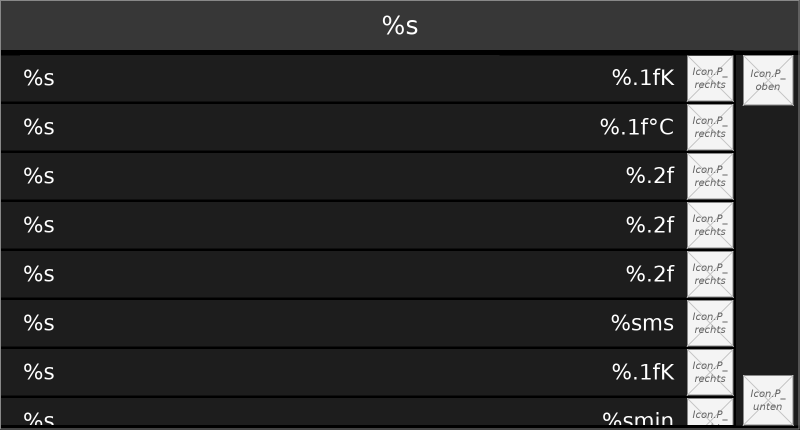
VISUALIZATION SW_WP_EEV_Liste  // 800x430
VAR_IN_OUT
	FB_EEV:EEV;	
	
END_VAR
	
VAR_INPUT
	i_Titel:INT;

END_VAR

VAR
	i_ref_versch:INT;
END_VAR
    Rectangle (0,0 800x50), "%s", text list: 'Sprachen', text index: i_Titel
    Rectangle (736,55 64x370)
    Image (743,375 50x50), image: Icon.P_unten
        OnMouseClick: execute { i_ref_versch:=i_ref_versch + 53; }
    Image (743,55 50x50), image: Icon.P_oben
        OnMouseClick: execute { i_ref_versch:=i_ref_versch - 53; }
    Group (0,50 733x590)
        p2738717112: i_ref_versch
        Rectangle (0,5 733x46)
        Rectangle (0,54 733x46)
        Rectangle (547,5 130x45), "%.1fK", text variable: FB_EEV.f_SollwertUBH
        Rectangle (547,54 130x46), "%.1f°C", text variable: FB_EEV.f_MOP
        Image (687,5 46x46), image: Icon.P_rechts
            OnMouseClick: execute { GWP_Library.Visu.i_Frame_Index:=1; }
        Image (687,54 46x46), image: Icon.P_rechts
            OnMouseClick: execute { GWP_Library.Visu.i_Frame_Index:=2; }
        Rectangle (0,103 733x46)
        Rectangle (0,152 733x46)
        Rectangle (0,201 733x46)
        Rectangle (0,250 733x46)
        Rectangle (0,299 733x46)
        Rectangle (0,348 733x46)
        Rectangle (0,397 733x46)
        Rectangle (0,446 733x46)
        Rectangle (0,495 733x46)
        Rectangle (547,103 130x45), "%.2f", text variable: FB_EEV.f_PFaktor
            OnMouseClick: execute { GWP_Library.Visu.i_Frame_Index:=2; }
        Rectangle (547,152 130x46), "%.2f", text variable: FB_EEV.f_IFaktor
        Rectangle (547,201 130x46), "%.2f", text variable: FB_EEV.f_DFaktor
        Rectangle (547,250 130x46), "%sms", text variable: FB_EEV.t_Takt.wMilliseconds
        Rectangle (547,299 130x46), "%.1fK", text variable: FB_EEV.f_MinUBH
        Rectangle (547,348 130x46), "%smin", text variable: FB_EEV.t_AL_EEV.wMinute
        Rectangle (547,446 130x46), "Ein"
        Rectangle (547,495 130x46), "Ein"
        Image (687,103 46x46), image: Icon.P_rechts
            OnMouseClick: execute { GWP_Library.Visu.i_Frame_Index:=3; }
        Image (687,495 46x46), image: Icon.P_rechts
        Image (687,446 46x46), image: Icon.P_rechts
        Image (687,397 46x46), image: Icon.P_rechts
            OnMouseClick: execute { GWP_Library.Visu.i_Frame_Index:=9; }
        Image (687,348 46x46), image: Icon.P_rechts
            OnMouseClick: execute { GWP_Library.Visu.i_Frame_Index:=8; }
        Image (687,299 46x46), image: Icon.P_rechts
            OnMouseClick: execute { GWP_Library.Visu.i_Frame_Index:=7; }
        Image (687,250 46x46), image: Icon.P_rechts
            OnMouseClick: execute { GWP_Library.Visu.i_Frame_Index:=6; }
        Image (687,201 46x46), image: Icon.P_rechts
            OnMouseClick: execute { GWP_Library.Visu.i_Frame_Index:=5; }
        Image (687,152 46x46), image: Icon.P_rechts
            OnMouseClick: execute { GWP_Library.Visu.i_Frame_Index:=4; }
        Rectangle (0,544 733x46)
        Rectangle (547,544 130x45), "Ein"
        Image (687,544 46x46), image: Icon.P_rechts
        Image (79,380 50x50), image: Icon.zurueck
            OnMouseClick:  Assign=Sollwertmenu_Waermegewinnung, Type=Assignment
            OnMouseClick: execute { i_verschieben:=0; }
        Rectangle (0,0 733x5)
        Rectangle (20,5 479x46), "%s", text list: 'Sprachen', text index: 85
        Rectangle (20,54 479x46), "%s", text list: 'Sprachen', text index: 86
        Rectangle (20,152 479x46), "%s", text list: 'Sprachen', text index: 88
        Rectangle (20,103 479x46), "%s", text list: 'Sprachen', text index: 87
        Rectangle (20,201 479x46), "%s", text list: 'Sprachen', text index: 89
        Rectangle (20,250 479x46), "%s", text list: 'Sprachen', text index: 90
        Rectangle (20,299 479x46), "%s", text list: 'Sprachen', text index: 91
        Rectangle (20,348 479x46), "%s", text list: 'Sprachen', text index: 92
        Rectangle (20,397 479x46), "%s", text list: 'Sprachen', text index: 72
        Rectangle (20,446 479x46), "%s", text list: 'Sprachen'
        Rectangle (20,495 479x46), "%s", text list: 'Sprachen'
        Rectangle (20,544 479x46), "%s", text list: 'Sprachen'
        Rectangle (0,375 733x5)
END_VISUALIZATION

// VISUs/Sollwertmenu_9/Wärmepumpe/Einsatzgrenzen/SW_WP_Einsatzgrenzen
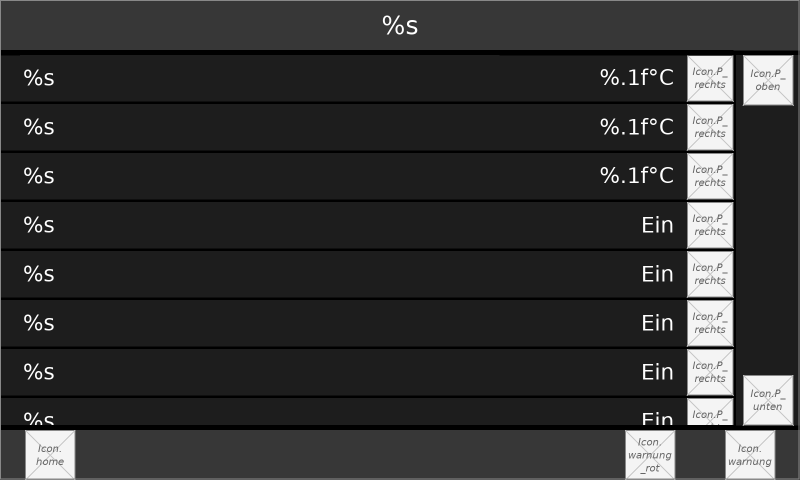
VISUALIZATION SW_WP_Einsatzgrenzen  // 800x480
VAR_IN_OUT
	FB_Einsatzgrenzen:Einsatzgrenzen;
END_VAR
    Frame (0,0 800x430)
        shows SW_WP_Einsatzgrenzen_Liste()
    Frame (0,430 800x50)
        shows Fusszeile_50()
END_VISUALIZATION

// VISUs/Sollwertmenu_9/Wärmepumpe/Einsatzgrenzen/SW_WP_Einsatzgrenzen_Liste
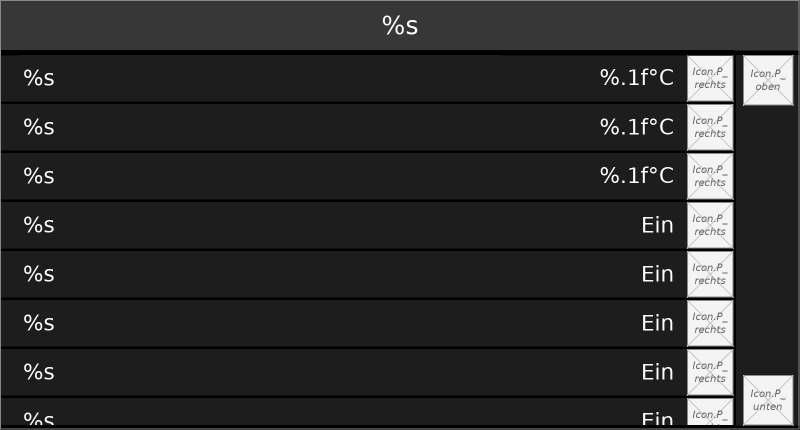
VISUALIZATION SW_WP_Einsatzgrenzen_Liste  // 800x430
VAR_IN_OUT
	FB_Einsatzgrenzen:Einsatzgrenzen;
END_VAR

VAR_INPUT
	i_Titel:INT;
END_VAR

VAR
	i_verschieben:INT;
 END_VAR
    Rectangle (0,55 733x46)
    Rectangle (0,104 733x46)
    Rectangle (547,55 130x45), "%.1f°C", text variable: FB_EEV.f_Regelsignal
    Rectangle (547,104 130x46), "%.1f°C"
    Image (687,55 46x46), image: Icon.P_rechts
        OnMouseClick: execute { GWP_Library.Visu.i_Frame_Index:=1; }
    Image (687,104 46x46), image: Icon.P_rechts
        OnMouseClick: execute { GWP_Library.Visu.i_Frame_Index:=2; }
    Rectangle (0,153 733x46)
    Rectangle (0,202 733x46)
    Rectangle (0,251 733x46)
    Rectangle (0,300 733x46)
    Rectangle (0,349 733x46)
    Rectangle (0,398 733x46)
    Rectangle (0,447 733x46)
    Rectangle (0,496 733x46)
    Rectangle (0,545 733x46)
    Rectangle (547,153 130x45), "%.1f°C"
        OnMouseClick: execute { GWP_Library.Visu.i_Frame_Index:=2; }
    Rectangle (547,202 130x46), "Ein"
    Rectangle (547,251 130x46), "Ein"
    Rectangle (547,300 130x46), "Ein"
    Rectangle (547,349 130x46), "Ein"
    Rectangle (547,447 130x46), "Ein"
    Rectangle (547,398 130x46), "Ein"
    Rectangle (547,496 130x46), "Ein"
    Rectangle (547,545 130x46), "Ein"
    Image (687,153 46x46), image: Icon.P_rechts
        OnMouseClick: execute { GWP_Library.Visu.i_Frame_Index:=3; }
    Image (687,545 46x46), image: Icon.P_rechts
    Image (687,496 46x46), image: Icon.P_rechts
    Image (687,447 46x46), image: Icon.P_rechts
    Image (687,398 46x46), image: Icon.P_rechts
    Image (687,349 46x46), image: Icon.P_rechts
    Image (687,300 46x46), image: Icon.P_rechts
    Image (687,251 46x46), image: Icon.P_rechts
    Image (687,202 46x46), image: Icon.P_rechts
    Rectangle (0,594 733x46)
    Rectangle (547,594 130x45), "Ein"
    Image (687,594 46x46), image: Icon.P_rechts
    Image (79,430 50x50), image: Icon.zurueck
        OnMouseClick:  Assign=Sollwertmenu_Waermegewinnung, Type=Assignment
        OnMouseClick: execute { i_verschieben:=0; }
    Rectangle (0,0 800x50), "%s", text list: 'Sprachen', text index: i_Titel
    Rectangle (736,55 64x370)
    Image (743,375 50x50), image: Icon.P_unten
        OnMouseClick: execute {
            IF i_verschieben<0 THEN
            	i_verschieben:=i_verschieben+53;
            End_if
        }
    Image (743,55 50x50), image: Icon.P_oben
        OnMouseClick: execute {
            IF  i_verschieben>-200 THEN
            	i_verschieben:=i_verschieben-53;
            End_if
        }
    Rectangle (0,50 733x5)
    Rectangle (20,55 479x46), "%s", text list: 'Sprachen'
    Rectangle (20,104 479x46), "%s", text list: 'Sprachen'
    Rectangle (20,202 479x46), "%s", text list: 'Sprachen'
    Rectangle (20,153 479x46), "%s", text list: 'Sprachen'
    Rectangle (20,251 479x46), "%s", text list: 'Sprachen'
    Rectangle (20,300 479x46), "%s", text list: 'Sprachen'
    Rectangle (20,349 479x46), "%s", text list: 'Sprachen'
    Rectangle (20,398 479x46), "%s", text list: 'Sprachen'
    Rectangle (20,447 479x46), "%s", text list: 'Sprachen'
    Rectangle (20,496 479x46), "%s", text list: 'Sprachen'
    Rectangle (20,545 479x46), "%s", text list: 'Sprachen'
    Rectangle (20,594 479x46), "%s", text list: 'Sprachen'
    Rectangle (0,425 733x5)
END_VISUALIZATION

// VISUs/Sollwertmenu_9/Wärmepumpe/Kachel_Allgemein
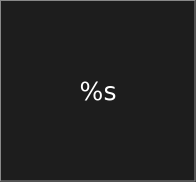
VISUALIZATION Kachel_Allgemein  // 196x182
    Rectangle (0,0 196x182), "%s", text list: 'Sprachen', text index: 18
END_VISUALIZATION

// VISUs/Sollwertmenu_9/Wärmepumpe/Kachel_EEV
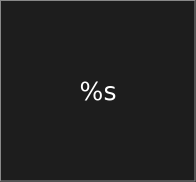
VISUALIZATION Kachel_EEV  // 196x182
    Rectangle (0,0 196x182), "%s", text list: 'Sprachen', text index: 15
END_VISUALIZATION

// VISUs/Sollwertmenu_9/Wärmepumpe/Kachel_Einsatzgrenzen
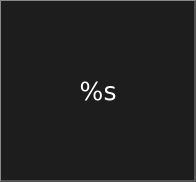
VISUALIZATION Kachel_Einsatzgrenzen  // 196x182
    Rectangle (0,0 196x182), "%s", text list: 'Sprachen', text index: 16
END_VISUALIZATION

// VISUs/Sollwertmenu_9/Wärmepumpe/Kachel_Verdichter
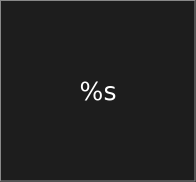
VISUALIZATION Kachel_Verdichter  // 196x182
    Rectangle (0,0 196x182), "%s", text list: 'Sprachen', text index: 17
END_VISUALIZATION

// VISUs/Sollwertmenu_9/Wärmepumpe/Sollwertmenu_Waermepumpe
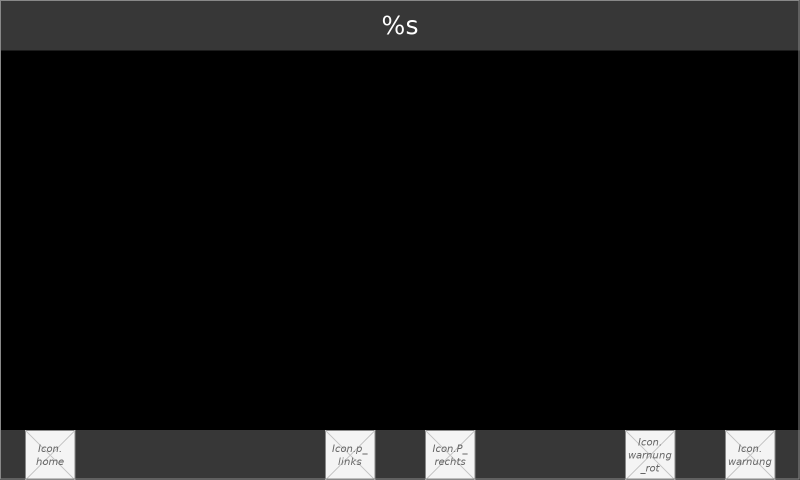
VISUALIZATION Sollwertmenu_Waermepumpe  // 800x480
VAR_IN_OUT
		
END_VAR

VAR
	i_verschieben:INT;

END_VAR
    Image (425,430 50x50), image: Icon.reinnavigieren
    Image (325,430 50x50), image: Icon.reinnavigieren
    Rectangle (0,0 800x50), "%s", text list: 'Sprachen', text index: 14
    Frame (0,430 800x50)
        shows Fusszeile_50()
    Image (425,430 50x50), image: Icon.P_rechts
        OnMouseClick: execute {
            IF i_verschieben>-800 THEN
            	i_verschieben:=i_verschieben-800;
            END_IF
        }
    Image (325,430 50x50), image: Icon.p_links
        OnMouseClick: execute {
            IF i_verschieben<0 THEN
            	i_verschieben:=i_verschieben+800;
            END_IF
        }
    Rectangle (88,515 454x57), "Kachel 1: 0;55 *** Kachel 2: 201;55 *** Kachel 3: 402;55 *** Kachel 4: 604;55 Kachel 5: 0;242 *** Kachel 6: 201;242 *** Kachel 7: 402;242 *** Kachel 8: 604;242"
END_VISUALIZATION

// VISUs/Sollwertmenu_9/Wärmesenke/Kachel_Heizgruppen
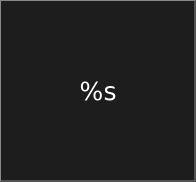
VISUALIZATION Kachel_Heizgruppen  // 196x182
    Rectangle (0,0 196x182), "%s", text list: 'Sprachen', text index: 23
END_VISUALIZATION

// VISUs/Sollwertmenu_9/Wärmesenke/Kachel_Hochhaltung
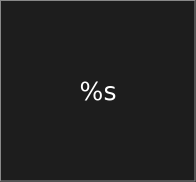
VISUALIZATION Kachel_Hochhaltung  // 196x182
    Rectangle (0,0 196x182), "%s", text list: 'Sprachen', text index: 24
END_VISUALIZATION

// VISUs/Sollwertmenu_9/Wärmesenke/Kachel_HWP
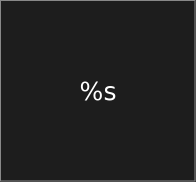
VISUALIZATION Kachel_HWP  // 196x182
    Rectangle (0,0 196x182), "%s", text list: 'Sprachen', text index: 21
END_VISUALIZATION

// VISUs/Sollwertmenu_9/Wärmesenke/Kachel_TWW
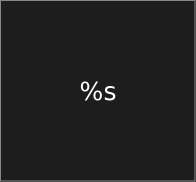
VISUALIZATION Kachel_TWW  // 196x182
    Rectangle (0,0 196x182), "%s", text list: 'Sprachen', text index: 22
END_VISUALIZATION

// VISUs/Sollwertmenu_9/Wärmesenke/Kachel_UWP_Verfl
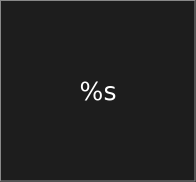
VISUALIZATION Kachel_UWP_Verfl  // 196x182
    Rectangle (0,0 196x182), "%s", text list: 'Sprachen', text index: 20
END_VISUALIZATION

// VISUs/Sollwertmenu_9/Wärmesenke/Sollwertmenu_Waermesenke
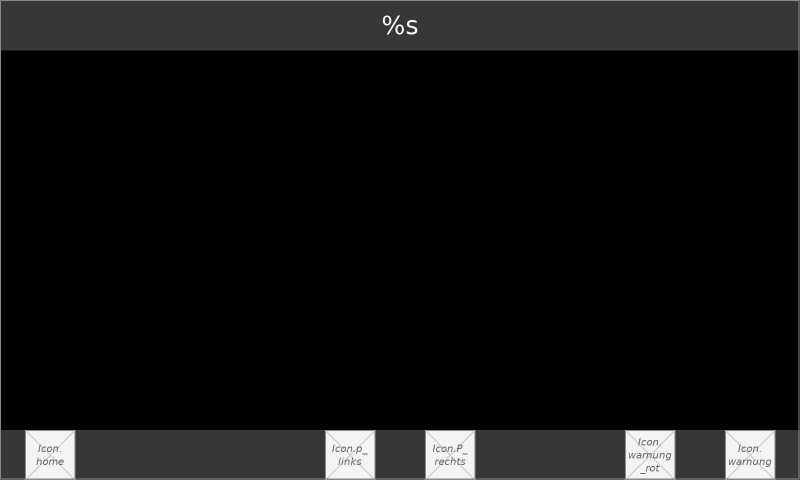
VISUALIZATION Sollwertmenu_Waermesenke  // 800x480
VAR_IN_OUT
		
END_VAR

VAR
	i_verschieben:INT;

END_VAR
    Image (425,430 50x50), image: Icon.reinnavigieren
    Image (325,430 50x50), image: Icon.reinnavigieren
    Rectangle (0,0 800x50), "%s", text list: 'Sprachen', text index: 19
    Frame (0,430 800x50)
        shows Fusszeile_50()
    Image (425,430 50x50), image: Icon.P_rechts
        OnMouseClick: execute {
            IF i_verschieben>-800 THEN
            	i_verschieben:=i_verschieben-800;
            END_IF
        }
    Image (325,430 50x50), image: Icon.p_links
        OnMouseClick: execute {
            IF i_verschieben<0 THEN
            	i_verschieben:=i_verschieben+800;
            END_IF
        }
    Rectangle (88,515 483x57), "Kachel 1: 0;55 *** Kachel 2: 201;55 *** Kachel 3: 402;55 *** Kachel 4: 604;55 Kachel 5: 0;242 *** Kachel 6: 201;242 *** Kachel 7: 402;242 *** Kachel 8: 604;242"
END_VISUALIZATION

// VISUs/Sprache/Spracheistellungen
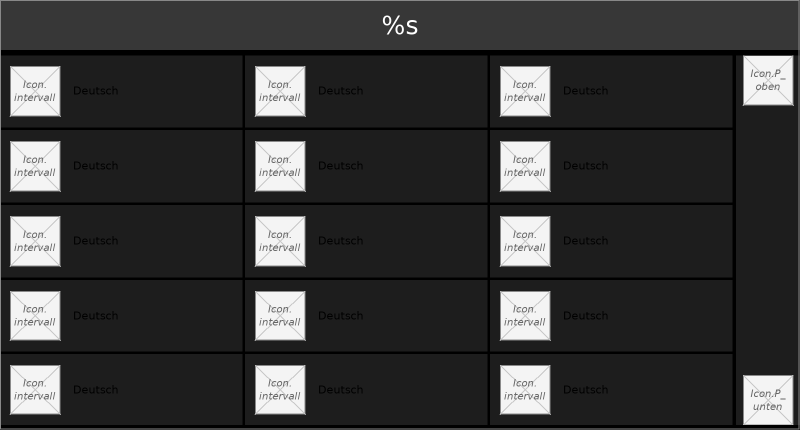
VISUALIZATION Spracheistellungen  // 800x430
VAR_IN_OUT

END_VAR

VAR_INPUT
	
END_VAR

VAR
	i_verschieben:INT;
 END_VAR
    Group (0,55 732x743)
        p2738717112: i_verschieben
        Rectangle (490,0 242x72)
        Rectangle (560,18 151x36), "Deutsch"
        Image (500,11 50x50), image: Icon.intervall
        Rectangle (245,0 242x72)
        Rectangle (315,18 151x36), "Deutsch"
        Image (255,11 50x50), image: Icon.intervall
        Rectangle (0,0 242x72)
        Rectangle (70,18 151x36), "Deutsch"
        Image (10,11 50x50), image: Icon.intervall
        Rectangle (490,75 242x72)
        Rectangle (560,93 151x36), "Deutsch"
        Image (500,86 50x50), image: Icon.intervall
        Rectangle (245,75 242x72)
        Rectangle (315,93 151x36), "Deutsch"
        Image (255,86 50x50), image: Icon.intervall
        Rectangle (0,75 242x72)
        Rectangle (70,93 151x36), "Deutsch"
        Image (10,86 50x50), image: Icon.intervall
        Rectangle (490,150 242x72)
        Rectangle (560,168 151x36), "Deutsch"
        Image (500,161 50x50), image: Icon.intervall
        Rectangle (245,150 242x72)
        Rectangle (315,168 151x36), "Deutsch"
        Image (255,161 50x50), image: Icon.intervall
        Rectangle (0,150 242x72)
        Rectangle (70,168 151x36), "Deutsch"
        Image (10,161 50x50), image: Icon.intervall
        Rectangle (490,225 242x71)
        Rectangle (560,243 151x36), "Deutsch"
        Image (500,236 50x49), image: Icon.intervall
        Rectangle (245,225 242x71)
        Rectangle (315,243 151x36), "Deutsch"
        Image (255,236 50x49), image: Icon.intervall
        Rectangle (0,225 242x71)
        Rectangle (70,243 151x36), "Deutsch"
        Image (10,236 50x49), image: Icon.intervall
        Rectangle (490,299 242x71)
        Rectangle (560,317 151x36), "Deutsch"
        Image (500,310 50x49), image: Icon.intervall
        Rectangle (245,299 242x71)
        Rectangle (315,317 151x36), "Deutsch"
        Image (255,310 50x49), image: Icon.intervall
        Rectangle (0,299 242x71)
        Rectangle (70,317 151x36), "Deutsch"
        Image (10,310 50x49), image: Icon.intervall
        Rectangle (490,373 242x72)
        Rectangle (560,391 151x36), "Deutsch"
        Image (500,384 50x50), image: Icon.intervall
        Rectangle (245,373 242x72)
        Rectangle (315,391 151x36), "Deutsch"
        Image (255,384 50x50), image: Icon.intervall
        Rectangle (0,373 242x72)
        Rectangle (70,391 151x36), "Deutsch"
        Image (10,384 50x50), image: Icon.intervall
        Rectangle (490,448 242x72)
        Rectangle (560,466 151x36), "Deutsch"
        Image (500,459 50x50), image: Icon.intervall
        Rectangle (245,448 242x72)
        Rectangle (315,466 151x36), "Deutsch"
        Image (255,459 50x50), image: Icon.intervall
        Rectangle (0,448 242x72)
        Rectangle (70,466 151x36), "Deutsch"
        Image (10,459 50x50), image: Icon.intervall
        Rectangle (490,523 242x72)
        Rectangle (560,541 151x36), "Deutsch"
        Image (500,534 50x50), image: Icon.intervall
        Rectangle (245,523 242x72)
        Rectangle (315,541 151x36), "Deutsch"
        Image (255,534 50x50), image: Icon.intervall
        Rectangle (0,523 242x72)
        Rectangle (70,541 151x36), "Deutsch"
        Image (10,534 50x50), image: Icon.intervall
        Rectangle (490,598 242x71)
        Rectangle (560,616 151x36), "Deutsch"
        Image (500,609 50x49), image: Icon.intervall
        Rectangle (245,598 242x71)
        Rectangle (315,616 151x36), "Deutsch"
        Image (255,609 50x49), image: Icon.intervall
        Rectangle (0,598 242x71)
        Rectangle (70,616 151x36), "Deutsch"
        Image (10,609 50x49), image: Icon.intervall
        Rectangle (490,672 242x71)
        Rectangle (560,690 151x36), "Deutsch"
        Image (500,683 50x49), image: Icon.intervall
        Rectangle (245,672 242x71)
        Rectangle (315,690 151x36), "Deutsch"
        Image (255,683 50x49), image: Icon.intervall
        Rectangle (0,672 242x71)
        Rectangle (70,690 151x36), "Deutsch"
        Image (10,683 50x49), image: Icon.intervall
    Rectangle (0,0 800x50), "%s", text list: 'Sprachen', text index: 70
    Group (736,55 64x370)
        Rectangle (0,0 64x370)
        Image (7,320 50x50), image: Icon.P_unten
            OnMouseClick: execute {
                IF i_verschieben<0 THEN
                	i_verschieben:=i_verschieben+75;
                End_if
            }
        Image (7,0 50x50), image: Icon.P_oben
            OnMouseClick: execute {
                IF  i_verschieben>-375 THEN
                	i_verschieben:=i_verschieben-75;
                End_if
            }
    Frame (0,430 800x50)
        shows Fusszeile_50()
    Rectangle (0,50 800x5)
    Rectangle (0,425 800x5)
END_VISUALIZATION

// VISUs/Zeitprogramm/EIn_Aus_Zeit_aendern
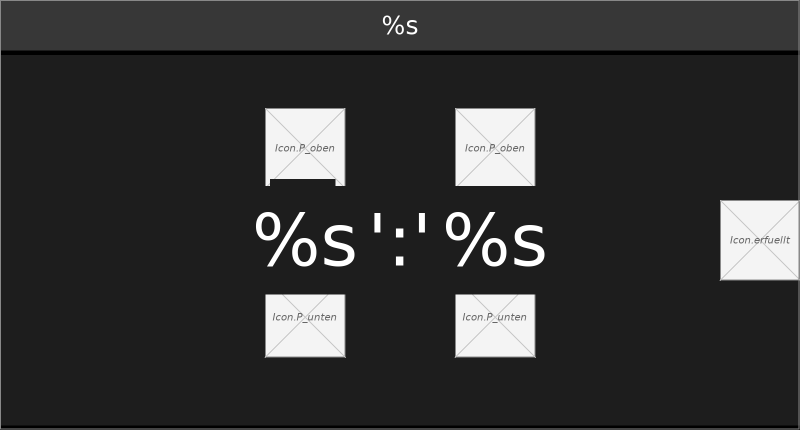
VISUALIZATION EIn_Aus_Zeit_aendern  // 800x430
VAR

END_VAR
VAR_IN_OUT
	f_Minuten:WORD;
	f_Stunden:WORD;	
END_VAR

VAR_INPUT
	i_titel:INT;
END_VAR
    Rectangle (0,0 800x50), "%s", text list: 'Sprachen', text index: i_titel
    Rectangle (0,55 800x370), text variable: f_Data
    Image (720,200 80x80), image: Icon.erfuellt
        OnMouseClick: execute { GWP_Library.Visu.i_Frame_Index:=0; }
    Image (265,108 80x80), image: Icon.P_oben
        OnMouseClick: execute { f_Stunden:=f_Stunden +1; }
    Image (455,108 80x80), image: Icon.P_oben
        OnMouseClick: execute { f_Minuten:=f_Minuten +1; }
    Image (265,277 80x80), image: Icon.P_unten
        OnMouseClick: execute { f_Stunden:=f_Stunden -1; }
    Image (455,277 80x80), image: Icon.P_unten
        OnMouseClick: execute { f_Minuten:=f_Minuten -1; }
    Rectangle (420,186 150x108), "%s", text variable: f_Minuten
    Rectangle (270,179 65x105)
    Rectangle (230,186 150x108), "%s", text variable: f_Stunden
    Rectangle (395,186 10x108), "':'"
END_VISUALIZATION

// VISUs/Zeitprogramm/Wochenuhr_W7
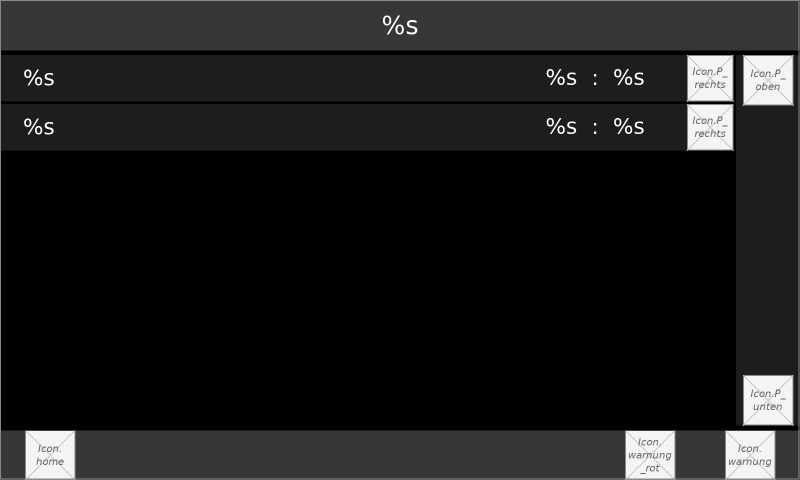
VISUALIZATION Wochenuhr_W7  // 800x480
VAR_IN_OUT
	FB_CLK_W7:CLK_W7;

END_VAR
    Frame (0,430 800x50)
        shows Fusszeile_50()
    Frame (0,0 800x430), frame switch variable: GWP_Library.Visu.i_Frame_Index
        shows Wochenuhr_W7_Liste(i_Titel := 52, FB_CLK_W7 := FB_CLK_W7)
        shows EIn_Aus_Zeit_aendern(i_titel := 68, f_Minuten := FB_CLK_W7.t_Ein_Mo.wMinute, f_Stunden := FB_CLK_W7.t_Ein_Mo.wHour)
        shows EIn_Aus_Zeit_aendern(i_titel := 68, f_Minuten := FB_CLK_W7.t_Aus_Mo.wMinute, f_Stunden := FB_CLK_W7.t_Aus_Mo.wHour)
END_VISUALIZATION

// VISUs/Zeitprogramm/Wochenuhr_W7_Liste
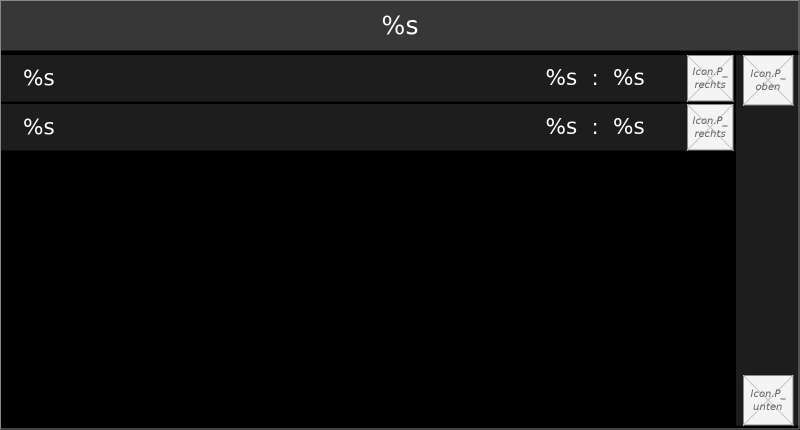
VISUALIZATION Wochenuhr_W7_Liste  // 800x430
VAR_IN_OUT
	FB_CLK_W7:CLK_W7;
	
END_VAR
VAR_INPUT
	i_Titel:INT;
END_VAR
    Rectangle (0,0 800x50), "%s", text list: 'Sprachen', text index: i_Titel
    Group (736,55 64x370)
        Rectangle (0,0 64x370)
        Image (7,320 50x50), image: Icon.P_unten
        Image (7,0 50x50), image: Icon.P_oben
    Rectangle (0,55 733x46)
    Image (687,55 46x46), image: Icon.P_rechts
        OnMouseClick: execute { GWP_Library.Visu.i_Frame_Index:=1; }
    Rectangle (610,55 70x45), "%s", text variable: FB_CLK_W7.t_Ein_Mo.wMinute
    Rectangle (510,55 70x45), "%s", text variable: FB_CLK_W7.t_Ein_Mo.wHour
    Rectangle (590,55 10x45), ":", text variable: FB_CLK_W7.t_Ein_Mo.wMinute
    Rectangle (20,55 400x46), "%s", text list: 'Sprachen', text index: 54
    Rectangle (0,104 733x46)
    Image (687,104 46x46), image: Icon.P_rechts
        OnMouseClick: execute { GWP_Library.Visu.i_Frame_Index:=2; }
    Rectangle (610,104 70x45), "%s", text variable: FB_CLK_W7.t_Aus_Mo.wMinute
    Rectangle (510,104 70x45), "%s", text variable: FB_CLK_W7.t_Aus_Mo.wHour
    Rectangle (590,104 10x45), ":", text variable: FB_CLK_W7.t_Ein_Mo.wMinute
    Rectangle (20,104 400x46), "%s", text list: 'Sprachen', text index: 55
END_VISUALIZATION

// VISUs/test_1
VISUALIZATION test_1  // 800x400
END_VISUALIZATION

(* text list Sprachen (id | default | Deutsch | Englisch | De)
  100 | Verzoegerung Stufe 2 |  |  | 
  101 | Verzögerung Stufe 1 |  |  | 
  0 | Wärmegewinnung |  |  | 
  1 | Wärmepumpe |  |  | 
  2 | Wärmesenke |  |  | 
  3 | Sollwertmenue |  |  | 
  4 | Sollwerte Wärmegewinnung |  |  | 
  5 | UWP Verd. |  |  | 
  6 | Erdsonde |  |  | 
  7 | Grundwasser |  |  | 
  8 | Luft |  |  | 
  9 | Tiefhaltung |  |  | 
  10 | Abtauspeicher |  |  | 
  11 | Abtauungen |  |  | 
  12 | Abwärme |  |  | 
  13 |  |  |  | 
  14 | Sollwerte Wärmepumpe |  |  | 
  15 | EEV |  |  | 
  16 | Einsatzgrenzen |  |  | 
  17 | Verdichter |  |  | 
  18 | Allgemein |  |  | 
  19 | Sollwerte Wärmesenke |  |  | 
  20 | UWP Verflüssiger |  |  | 
  21 | HWP |  |  | 
  22 | TWW |  |  | 
  23 | Heizgruppe |  |  | 
  24 | Hochhaltung |  |  | 
  25 | Sollwerte UWP Verflüssiger |  |  | 
  26 | Sollwerte Erdsonden |  |  | 
  27 | Sollwerte Luft |  |  | 
  28 | Sollwerte Abwärme |  |  | 
  29 | Sollwerte Tiefhaltung |  |  | 
  30 | Sollwertänderung  |  |  | 
  31 | Infoseite |  |  | 
  32 | Hauptmenü |  |  | 
  33 | Sprachen |  |  | 
  34 | Login |  |  | 
  35 | Sollwerte |  |  | 
  36 | Verlaufs- diagramm |  |  | 
  37 | Uhrzeit einstellen |  |  | 
  38 | IBN |  |  | 
  39 | Konfiguration |  |  | 
  40 | Kontakt |  |  | 
  41 | Ein/Aus Wärmepumpe |  |  | 
  42 | Ein |  |  | 
  43 | Aus |  |  | 
  44 | IO-Auswahl |  |  | 
  45 | Digitale Eingänge |  |  | 
  46 | Digitale Ausgänge |  |  | 
  47 | Analoge Eingänge |  |  | 
  48 | Analoge Ausgänge |  |  | 
  49 | Status |  |  | 
  50 | Offset |  |  | 
  51 | Istwert |  |  | 
  52 | Wochenschaltuhr |  |  | 
  53 | Start Zeit |  |  | 
  5000 | Alarme |  |  | 
  54 | Montag Ein |  |  | 
  55 | Montag Aus |  |  | 
  56 | Dienstag Ein |  |  | 
  57 | Dienstag Aus |  |  | 
  58 | Mittwoch Ein |  |  | 
  59 | Mittwoch Aus |  |  | 
  60 | Donnerstag EIn |  |  | 
  61 | Donnerstag Aus |  |  | 
  62 | Freitag Ein |  |  | 
  63 | Freitag Aus |  |  | 
  64 | Samstag Ein |  |  | 
  65 | Samstag Aus |  |  | 
  66 | Sonntag Ein |  |  | 
  67 | Sonntag Aus |  |  | 
  68 | Ein-/Ausschaltzeit ändern |  |  | 
  69 | Sollwertänderung |  |  | 
  70 | Sprach Auswahl |  |  | 
  71 | Heizkurve |  |  | 
  84 | Dynamischer MOP |  |  | 
  85 | Sollwert Überhitzung |  |  | 
  86 | Maximaler Operating Pressure |  |  | 
  87 | P-Faktor für Regelung |  |  | 
  88 | I-Faktor für Regelung |  |  | 
  89 | D-Faktor für Regelung |  |  | 
  90 | Berechnungstakt PID Regler |  |  | 
  91 | Minimale Überhitzung |  |  | 
  92 | Zeit bis Alarm ausgelöst wird |  |  | 
  96 | Sollwerte EEV |  |  | 
  73 | Abbrechen |  |  | 
  72 | Sollwerte zurücksetzen |  |  | 
   |  |  |  |  *)
